// Mitsubishi GX Works2 project: GT_EX4   PLC: Q03UDV

PROGRAM MAIN
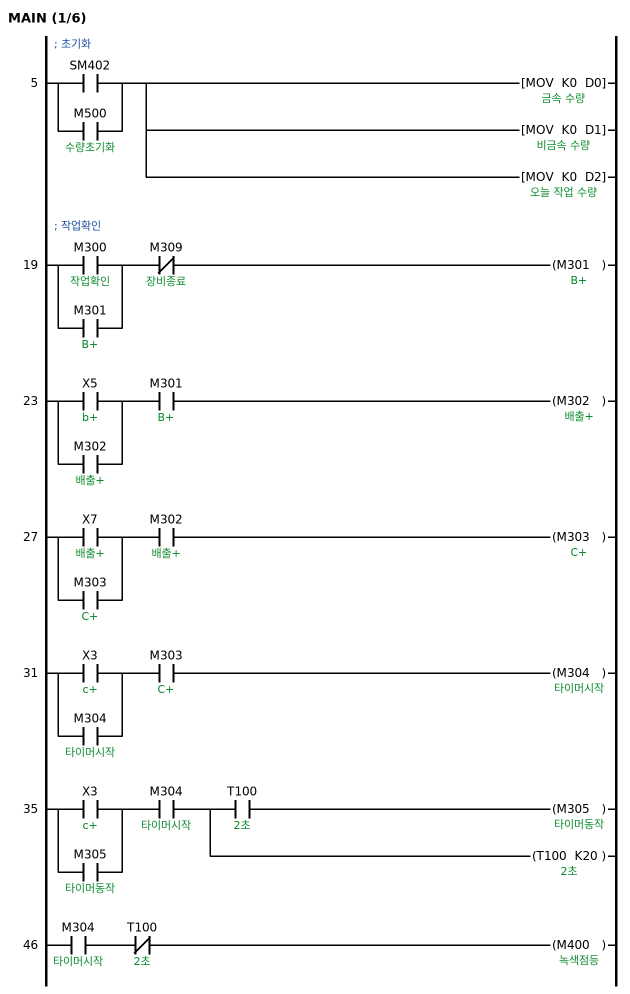
; 초기화
5     LD      SM402
      OR      M500  ; 수량초기화
      MOV     K0 D0  ; 금속 수량
      MOV     K0 D1  ; 비금속 수량
      MOV     K0 D2  ; 오늘 작업 수량
; 작업확인
19    LD      M300  ; 작업확인
      OR      M301  ; B+
      ANI     M309  ; 장비종료
      OUT     M301  ; B+
23    LD      X5  ; b+
      OR      M302  ; 배출+
      AND     M301  ; B+
      OUT     M302  ; 배출+
27    LD      X7  ; 배출+
      OR      M303  ; C+
      AND     M302  ; 배출+
      OUT     M303  ; C+
31    LD      X3  ; c+
      OR      M304  ; 타이머시작
      AND     M303  ; C+
      OUT     M304  ; 타이머시작
35    LD      X3  ; c+
      OR      M305  ; 타이머동작
      AND     M304  ; 타이머시작
      MPS
      AND     T100  ; 2초
      OUT     M305  ; 타이머동작
      MPP
      OUT     T100 K20  ; 2초
46    LD      M304  ; 타이머시작
      ANI     T100  ; 2초
      OUT     M400  ; 녹색점등
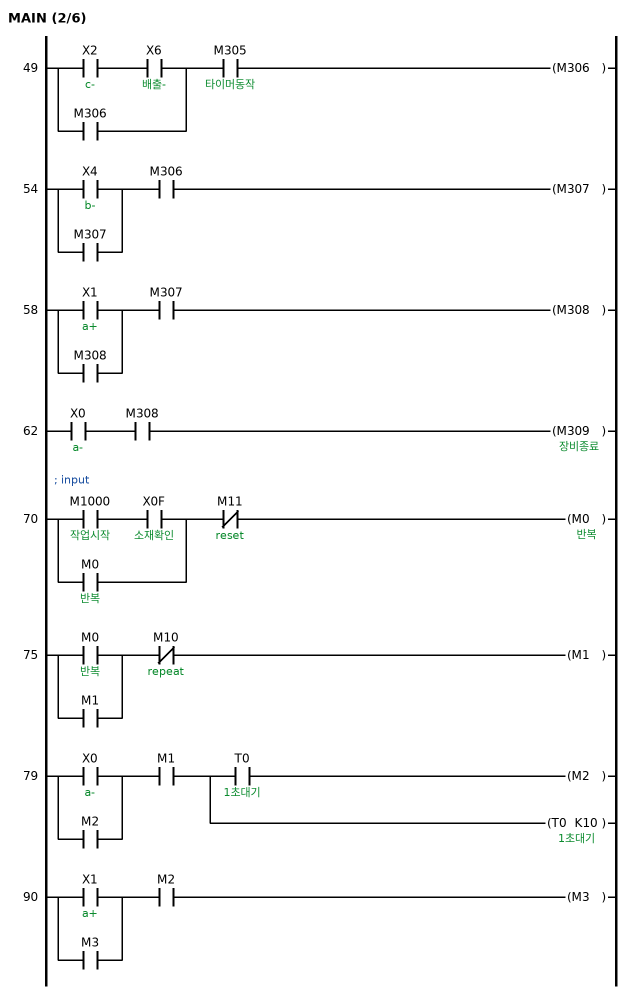
49    LD      X2  ; c-
      AND     X6  ; 배출-
      OR      M306
      AND     M305  ; 타이머동작
      OUT     M306
54    LD      X4  ; b-
      OR      M307
      AND     M306
      OUT     M307
58    LD      X1  ; a+
      OR      M308
      AND     M307
      OUT     M308
62    LD      X0  ; a-
      AND     M308
      OUT     M309  ; 장비종료
; input
70    LD      M1000  ; 작업시작
      AND     X0F  ; 소재확인
      OR      M0  ; 반복
      ANI     M11  ; reset
      OUT     M0  ; 반복
75    LD      M0  ; 반복
      OR      M1
      ANI     M10  ; repeat
      OUT     M1
79    LD      X0  ; a-
      OR      M2
      AND     M1
      MPS
      AND     T0  ; 1초대기
      OUT     M2
      MPP
      OUT     T0 K10  ; 1초대기
90    LD      X1  ; a+
      OR      M3
      AND     M2
      OUT     M3
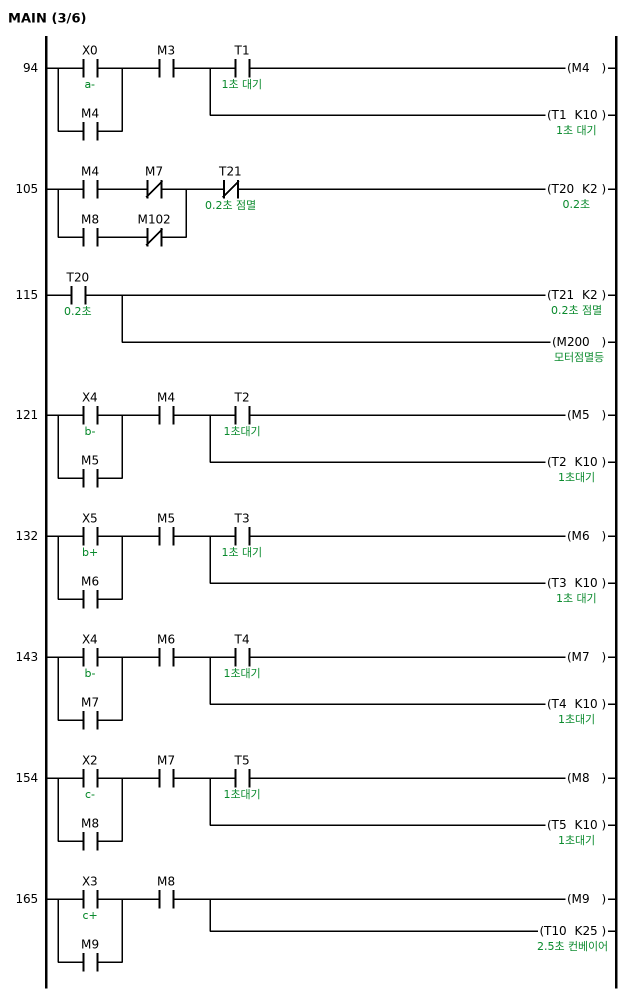
94    LD      X0  ; a-
      OR      M4
      AND     M3
      MPS
      AND     T1  ; 1초 대기
      OUT     M4
      MPP
      OUT     T1 K10  ; 1초 대기
105   LD      M4
      ANI     M7
      LD      M8
      ANI     M102
      ORB
      ANI     T21  ; 0.2초 점멸
      OUT     T20 K2  ; 0.2초
115   LD      T20  ; 0.2초
      OUT     T21 K2  ; 0.2초 점멸
      OUT     M200  ; 모터점멸등
121   LD      X4  ; b-
      OR      M5
      AND     M4
      MPS
      AND     T2  ; 1초대기
      OUT     M5
      MPP
      OUT     T2 K10  ; 1초대기
132   LD      X5  ; b+
      OR      M6
      AND     M5
      MPS
      AND     T3  ; 1초 대기
      OUT     M6
      MPP
      OUT     T3 K10  ; 1초 대기
143   LD      X4  ; b-
      OR      M7
      AND     M6
      MPS
      AND     T4  ; 1초대기
      OUT     M7
      MPP
      OUT     T4 K10  ; 1초대기
154   LD      X2  ; c-
      OR      M8
      AND     M7
      MPS
      AND     T5  ; 1초대기
      OUT     M8
      MPP
      OUT     T5 K10  ; 1초대기
165   LD      X3  ; c+
      OR      M9
      AND     M8
      OUT     M9
      OUT     T10 K25  ; 2.5초 컨베이어
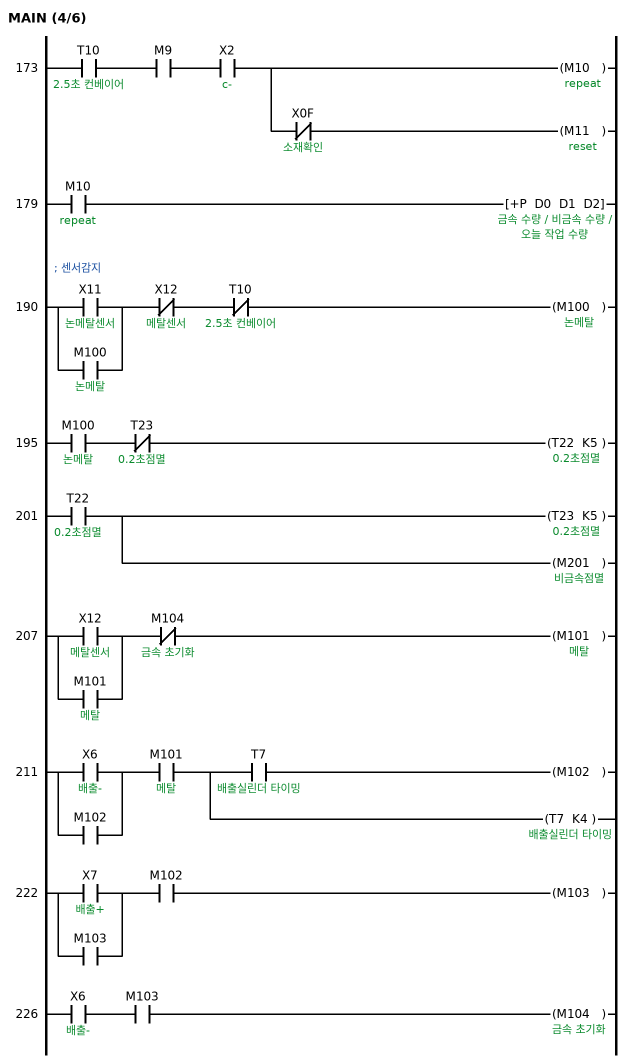
173   LD      T10  ; 2.5초 컨베이어
      AND     M9
      AND     X2  ; c-
      OUT     M10  ; repeat
      ANI     X0F  ; 소재확인
      OUT     M11  ; reset
179   LD      M10  ; repeat
      +P      D0 D1 D2
; 센서감지
190   LD      X11  ; 논메탈센서
      OR      M100  ; 논메탈
      ANI     X12  ; 메탈센서
      ANI     T10  ; 2.5초 컨베이어
      OUT     M100  ; 논메탈
195   LD      M100  ; 논메탈
      ANI     T23  ; 0.2초점멸
      OUT     T22 K5  ; 0.2초점멸
201   LD      T22  ; 0.2초점멸
      OUT     T23 K5  ; 0.2초점멸
      OUT     M201  ; 비금속점멸
207   LD      X12  ; 메탈센서
      OR      M101  ; 메탈
      ANI     M104  ; 금속 초기화
      OUT     M101  ; 메탈
211   LD      X6  ; 배출-
      OR      M102
      AND     M101  ; 메탈
      MPS
      AND     T7  ; 배출실린더 타이밍
      OUT     M102
      MPP
      OUT     T7 K4  ; 배출실린더 타이밍
222   LD      X7  ; 배출+
      OR      M103
      AND     M102
      OUT     M103
226   LD      X6  ; 배출-
      AND     M103
      OUT     M104  ; 금속 초기화
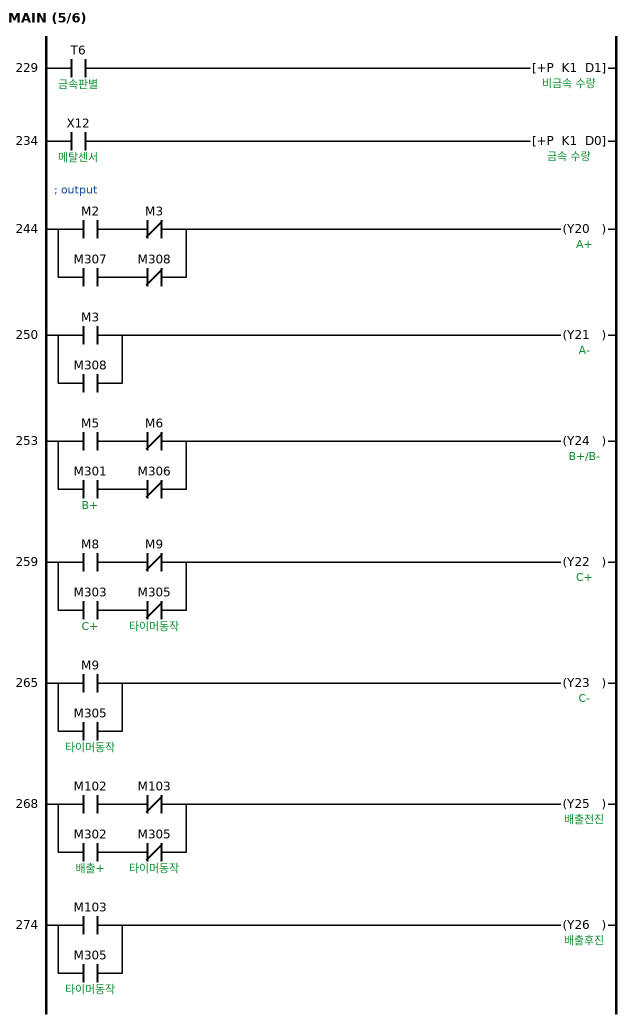
229   LD      T6  ; 금속판별
      +P      K1 D1
234   LD      X12  ; 메탈센서
      +P      K1 D0
; output
244   LD      M2
      ANI     M3
      LD      M307
      ANI     M308
      ORB
      OUT     Y20  ; A+
250   LD      M3
      OR      M308
      OUT     Y21  ; A-
253   LD      M5
      ANI     M6
      LD      M301  ; B+
      ANI     M306
      ORB
      OUT     Y24  ; B+/B-
259   LD      M8
      ANI     M9
      LD      M303  ; C+
      ANI     M305  ; 타이머동작
      ORB
      OUT     Y22  ; C+
265   LD      M9
      OR      M305  ; 타이머동작
      OUT     Y23  ; C-
268   LD      M102
      ANI     M103
      LD      M302  ; 배출+
      ANI     M305  ; 타이머동작
      ORB
      OUT     Y25  ; 배출전진
274   LD      M103
      OR      M305  ; 타이머동작
      OUT     Y26  ; 배출후진
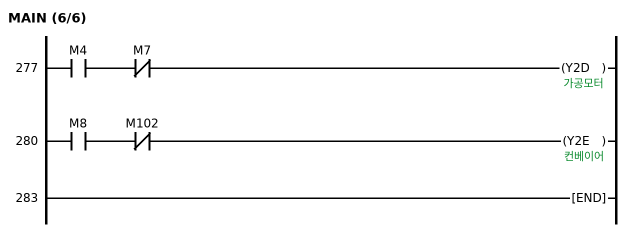
277   LD      M4
      ANI     M7
      OUT     Y2D  ; 가공모터
280   LD      M8
      ANI     M102
      OUT     Y2E  ; 컨베이어
283   END
END_PROGRAM
